Staubli VAL3: francais.dtx

public string No = "Non"
public string Yes = "Oui"
